# EPICS substitutions: db/ecmcEK1110.substitutions
file ecmcEcSlave.template
{
    pattern {}
            {}
}
